// TIA Portal V19 export
FUNCTION "Box Handler Simulation Logic" : Void   // FC20, LAD
{ S7_Optimized_Access := 'TRUE' }
// stored: AutoNumber false, SetENOAutomatically false
   VAR_TEMP
      ArmOn : Bool;
      ArmSpeed : Real;
   END_VAR
   VAR_TEMP   // added for the SCL form of the ladder/FBD networks
      _w1 : Bool;
      _w2 : Bool;
      _w3 : Bool;
   END_VAR
BEGIN

REGION Network 1: HMI Conveyor control logic
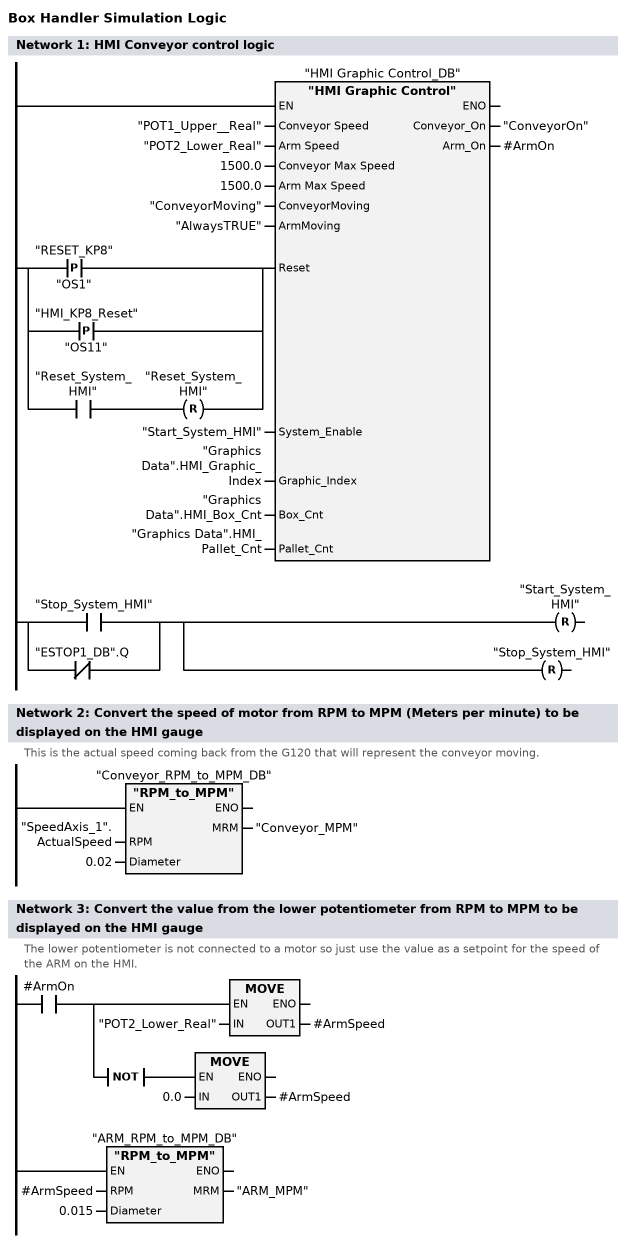
   RUNG wire#powerrail
      "HMI Graphic Control_DB"(Reset := wire#w1, "Conveyor Speed" := "POT1_Upper__Real", "Arm Speed" := "POT2_Lower_Real", "Conveyor Max Speed" := 1500.0, "Arm Max Speed" := 1500.0, ConveyorMoving := "ConveyorMoving", ArmMoving := "AlwaysTRUE", System_Enable := "Start_System_HMI", Graphic_Index := "Graphics Data".HMI_Graphic_Index, Box_Cnt := "Graphics Data".HMI_Box_Cnt, Pallet_Cnt := "Graphics Data".HMI_Pallet_Cnt, Conveyor_On => "ConveyorOn", Arm_On => #ArmOn)
   END_RUNG
   RUNG wire#powerrail
      P_Contact(operand := "RESET_KP8", bit := "OS1")
   END_RUNG wire#w1
   RUNG wire#powerrail
      P_Contact(operand := "HMI_KP8_Reset", bit := "OS11")
   END_RUNG wire#w1
   RUNG wire#powerrail
      Contact( "Reset_System_HMI" )
      R_Coil( "Reset_System_HMI" )
   END_RUNG wire#w1
   RUNG wire#powerrail
      Contact( "Stop_System_HMI" )
      wire#w2
      R_Coil( "Start_System_HMI" )
   END_RUNG
   RUNG wire#powerrail
      I_Contact( "ESTOP1_DB".Q )
   END_RUNG wire#w2
   RUNG wire#w2
      R_Coil( "Stop_System_HMI" )
   END_RUNG
   // the same network as SCL:
   #_w1 := "RESET_KP8" AND NOT "OS1";   // rising edge of "RESET_KP8"
   "OS1" := "RESET_KP8";
   #_w2 := "HMI_KP8_Reset" AND NOT "OS11";   // rising edge of "HMI_KP8_Reset"
   "OS11" := "HMI_KP8_Reset";
   #_w3 := "Reset_System_HMI";
   IF #_w3 THEN "Reset_System_HMI" := FALSE; END_IF;
   "HMI Graphic Control_DB"("Conveyor Speed" := "POT1_Upper__Real",   // "HMI Graphic Control"
                           "Arm Speed" := "POT2_Lower_Real",
                           "Conveyor Max Speed" := 1500.0,
                           "Arm Max Speed" := 1500.0,
                           ConveyorMoving := "ConveyorMoving",
                           ArmMoving := "AlwaysTRUE",
                           Reset := #_w1 OR #_w2 OR #_w3,
                           System_Enable := "Start_System_HMI",
                           Graphic_Index := "Graphics Data".HMI_Graphic_Index,
                           Box_Cnt := "Graphics Data".HMI_Box_Cnt,
                           Pallet_Cnt := "Graphics Data".HMI_Pallet_Cnt,
                           Conveyor_On => "ConveyorOn",
                           Arm_On => #ArmOn);
   IF "Stop_System_HMI" OR NOT "ESTOP1_DB".Q THEN
       "Start_System_HMI" := FALSE;
       "Stop_System_HMI" := FALSE;
   END_IF;
END_REGION

REGION Network 2: Convert the speed of motor from RPM to MPM (Meters per minute) to be displayed on the HMI gauge
   // This is the actual speed coming back from the G120 that will represent the conveyor moving.
   RUNG wire#powerrail
      "Conveyor_RPM_to_MPM_DB"(RPM := "SpeedAxis_1".ActualSpeed, Diameter := 0.02, MRM => "Conveyor_MPM")
   END_RUNG
   // the same network as SCL:
   "Conveyor_RPM_to_MPM_DB"(RPM := "SpeedAxis_1".ActualSpeed, Diameter := 0.02, MRM => "Conveyor_MPM");   // "RPM_to_MPM"
END_REGION

REGION Network 3: Convert the value from the lower potentiometer from RPM to MPM to be displayed on the HMI gauge
   // The lower potentiometer is not connected to a motor so just use the value as a setpoint for the speed of the ARM on the HMI.
   RUNG wire#powerrail
      Contact( #ArmOn )
      wire#w1
      Move(in := "POT2_Lower_Real", out1 => #ArmSpeed)
   END_RUNG
   RUNG wire#w1
      Not()
      Move(in := 0.0, out1 => #ArmSpeed)
   END_RUNG
   RUNG wire#powerrail
      "ARM_RPM_to_MPM_DB"(RPM := #ArmSpeed, Diameter := 0.015, MRM => "ARM_MPM")
   END_RUNG
   // the same network as SCL:
   IF #ArmOn THEN #ArmSpeed := "POT2_Lower_Real"; END_IF;
   IF NOT #ArmOn THEN #ArmSpeed := 0.0; END_IF;
   "ARM_RPM_to_MPM_DB"(RPM := #ArmSpeed, Diameter := 0.015, MRM => "ARM_MPM");   // "RPM_to_MPM"
END_REGION
END_FUNCTION
